(* IEC 61131-3 sources: Temperature-Cabinet-Control-Automation/codesys modbus proof of concept and test logs/src/POUs, 2 files *)

(* ---- PLC_PRG.st ---- *)
(*
    PROGRAM:  PLC_PRG
    Project:  Temperature Cabinet Setpoint Control from CODESYS HMI
    Author:   OJ (Omkar Joshi) - Oliver Mechatronics
    Language: IEC 61131-3 Structured Text (CODESYS 3.5, WebVisu)

    Cyclic entry point (MainTask). Instantiates the supervisory setpoint
    controller. Because FB_CabinetSetpointControl reads/writes GVL_Modbus
    and GVL_HMI directly in its body (see that FB's header note), this
    program only needs to pass through the operator-facing parameters
    and the safety interlock input.

    Matches the Project Development Package spec (Details A) and the
    build guide already in codesys modbus com port investigation and troubleshooting log/README.md.

    TODO (flagged in the Project Development Package, not yet resolved):
    xOverTempDI below is wired to GVL_Modbus.xModbusError as a
    placeholder. REPLACE with the real mapped EL1409 digital-input
    channel (spare over-temperature lamp contact) in the EtherCAT I/O
    mapping before relying on this interlock.
*)
PROGRAM PLC_PRG
VAR
    fbSetpoint : FB_CabinetSetpointControl;
END_VAR

(* ---- Drive the supervisory setpoint controller ---- *)
fbSetpoint(
    rRequestedSetpoint := GVL_HMI.rReqSetpoint,
    xSetCommand        := GVL_HMI.xSetBtn,
    xReset             := GVL_HMI.xResetBtn,
    xOverTempDI        := GVL_Modbus.xModbusError,  (* REPLACE with mapped EL1409 DI channel *)
    rMinSetpoint       := -40.0,
    rMaxSetpoint       := 200.0
);

(* ---- Consume dialog button one-shots ---- *)
GVL_HMI.xSetBtn   := FALSE;
GVL_HMI.xResetBtn := FALSE;

(* ---- PLC_PRG_TCP.st ---- *)
PROGRAM PLC_PRG
(* ======================================================================
   Retargeted for TCP register sources (Python gateway via Modbus TCP)
   ======================================================================
   Serial device abandoned. All reads/writes now come via the TCP slave
   device on the Modbus TCP master branch of the device tree.

   Proven register map (TCP holding registers, x10 integers):
     reg2 = chamber temperature (read-only, cyclic)
     reg3 = confirmed setpoint read-back (read-only, cyclic)
     reg4 = status/fault code (read-only, cyclic)
     reg0 = requested setpoint (write, cyclic or rising)
     reg1 = apply trigger (write, rising edge)

   I/O Mapping binds these to GVL_Modbus:
     reg2 -> wInput1Value (temperature)
     reg3 -> wSetpoint1Read (confirmed SP)
     reg4 -> wStatus (fault code: 0=OK, 2=WRITE_FAILED, 3=NOT_ACCEPTED, 4=RANGE, 5=COMMS)
     reg0 -> wSetpoint1Write (requested SP, x10)
     reg1 -> xWriteTrigger (apply pulse, BOOL as WORD 0/1)

   The state machine logic is unchanged from the serial version. Only the
   data sources changed: TCP channels instead of serial channels.
   ====================================================================== *)

VAR
    rChamberTemp        : REAL;
    rReqSetpoint        : REAL := 26.5;           (* set in watch window or WebVisu *)
    rConfirmedSetpoint  : REAL;

    rMinSetpoint        : REAL := -40.0;
    rMaxSetpoint        : REAL := 200.0;

    eSetpointState      : E_SetpointState := E_SetpointState.IDLE;
    eFaultCode          : E_FaultCode := E_FaultCode.NO_FAULT;

    xStartWrite         : BOOL := FALSE;          (* rising-edge trigger for manual test *)
    xPrevStartWrite     : BOOL := FALSE;
    xWriteTriggered     : BOOL := FALSE;

    dwWriteTimeout      : DWORD := 0;
    (* Must exceed the WORST-CASE confirm chain, not the typical one:
         gateway poll period            1.0 s   (POLL_PERIOD)
       + gateway RTU confirm read-back  0.5 s   (READ_TIMEOUT)
       + CODESYS cyclic read of reg3    2.0 s   (channel 3 trigger interval)
       = 3.5 s worst case, against a 3.0 s timeout -> spurious NOT_ACCEPTED on
       a write the F4S had actually taken. Raised to 10 s so only a genuine
       failure trips it; the gateway's own status codes (2/3/5) still fault
       fast, so a real rejection is never delayed by this headroom. *)
    dwMaxTimeout        : DWORD := 1000;          (* ~10s at 10ms MainTask *)

    dtNow               : DT;                      (* current local time for schedule *)
    uliHighRes          : ULINT;                   (* high-resolution time, raw ms since epoch, UTC *)
END_VAR

(* --- STEP 0: Cabinet on/off - EL2869 CH15/CH16 -> Omron CPM1A digital inputs ---
   AS-BUILT 6 Aug 2026 (README §19), supersedes the §17 F4-DI ramp gate for on/off.
   CH15 -> wire 102 -> Omron 0CH.00 (start input to the Omron's own start-stop-hold
   ladder logic). CH16 -> wire 103 -> Omron 0CH.01 (stop input). EL2869 DO GND is
   bonded to Omron COM0.

   xStartPulse and xStopPermit are plain, independently-commanded levels -- no
   timer, no derived pulse, no anti-short-cycle lockout. Set them from the watch
   window (or, later, WebVisu) and they hold until changed. The Omron's own
   program does the actual start-stop-hold latching, so CODESYS only needs to
   present a level on each input; it does not need to shape a pulse width the way
   the earlier (§15 Option C-era) design did.

   That earlier design drove xStartPulse off a TP one-shot fired on the rising
   edge of xStopPermit, modelling CH16 as a continuous 24 V supply that CH15
   briefly "pressed" through (the button-station supply-lift model). That model
   does not apply to the Omron's digital inputs and is what produced the reported
   "stop permit true, then false, then start pulse fires" sequence -- an artifact
   of the old coupling, not the Omron's behaviour. Removed here.

   The only guard kept in is stop-priority mutual exclusion: if both are ever
   commanded TRUE together, stop wins. This costs one line and there is no
   scenario where firing both at once is the intended action -- flag it for
   removal if that turns out to be unwanted.

   xCabinetOnCmd (scheduler-derived, below) is NOT wired into xStartPulse/
   xStopPermit yet -- open question, README §19, on whether the schedule should
   auto-drive start/stop or these should stay purely operator/CODESYS-commanded. *)
SysTimeRtcHighResGet(uliHighRes);
dtNow := ULINT_TO_DT(uliHighRes / 1000 + DINT_TO_ULINT(GVL_HMI.diUtcOffsetSec));  (* ms -> s, then UTC -> local *)

GVL_HMI.xCabinetOnCmd := NOT (GVL_HMI.xSchedEnable AND (dtNow < GVL_HMI.dtSchedStart));

IF GVL_HMI.xStopPermit THEN
    GVL_HMI.xStartPulse := FALSE;
END_IF

GVL_HMI.xCabinetRunning := GVL_HMI.xStartPulse AND NOT GVL_HMI.xStopPermit;  (* commanded-state
    proxy for WebVisu -- no independent run feedback wired back from the Omron yet, README §19.6 *)

(* --- STEP 0b: Front-panel keypad lock (§17/§18 F4 digital input design) ---
   NOT CURRENTLY WIRED. CH16 is now committed to the Omron stop input above, so
   xPanelLock has no live output channel until §18's D/I 2 is reallocated to a
   spare EL2869 channel (README §19.5). Left commented out rather than deleted so
   the logic is ready to reconnect once that channel is chosen and mapped:

   GVL_HMI.xPanelLock := GVL_HMI.xPanelLockCmd;
*)

(* --- STEP 1: Scale raw TCP values -> engineering units ---
   TCP registers carry x10 integers; we work in real degrees.
   All three reads come from the TCP channels (wInput1Value, wSetpoint1Read, wStatus).

   The registers carry SIGNED x10 integers in two's complement. WORD is an
   UNSIGNED type in IEC 61131-3, so dividing it directly turns -1.0 degC
   (raw 16#FFF6) into 6552.6 instead of -1.0. Every sub-zero temperature and
   every negative setpoint read-back was wrong, and the CONFIRM comparison
   below could never match one. WORD_TO_INT reinterprets the bit pattern as
   the signed value the F4S actually sent.
*)
rChamberTemp       := WORD_TO_INT(GVL_Modbus.wInput1Value)  / 10.0;
rConfirmedSetpoint := WORD_TO_INT(GVL_Modbus.wSetpoint1Read) / 10.0;

(* --- STEP 2: Detect rising edge on the manual test trigger ---
   When testing from watch window, toggle xStartWrite from FALSE to TRUE.
   In production (WebVisu or SCADA), the operator triggers via a button that
   sets a HMI variable, but the edge logic is the same.
*)
xWriteTriggered := (xStartWrite AND NOT xPrevStartWrite);
xPrevStartWrite := xStartWrite;

(* --- STEP 3: State machine (unchanged logic, TCP-based register sources) --- *)

CASE eSetpointState OF

    E_SetpointState.IDLE:
        (* Waiting for a write request. Hold the apply trigger low. *)
        GVL_Modbus.xWriteTrigger := FALSE;
        dwWriteTimeout := 0;

        IF xWriteTriggered THEN
            eSetpointState := E_SetpointState.READY;
        END_IF

    E_SetpointState.READY:
        (* Validate the requested setpoint against limits. *)
        IF rReqSetpoint < rMinSetpoint THEN
            eFaultCode := E_FaultCode.RANGE_LOW;
            eSetpointState := E_SetpointState.FAULTED;

        ELSIF rReqSetpoint > rMaxSetpoint THEN
            eFaultCode := E_FaultCode.RANGE_HIGH;
            eSetpointState := E_SetpointState.FAULTED;

        ELSE
            (* Valid range. Stage the request (x10 int) into the TCP write register.

               REAL_TO_DWORD is UNDEFINED for negative operands in IEC 61131-3
               -- it happened to produce the right bit pattern on this runtime,
               but that is luck, not contract, and it truncates instead of
               rounding (26.45 -> 264, not 265). REAL_TO_INT rounds and is
               defined across the whole -40..200 range; INT_TO_WORD then
               reinterprets the signed value as the two's-complement WORD the
               gateway expects on the wire. *)
            GVL_Modbus.wSetpoint1Write := INT_TO_WORD(REAL_TO_INT(rReqSetpoint * 10.0));
            eSetpointState := E_SetpointState.WRITING;
        END_IF

    E_SetpointState.WRITING:
        (* Pulse the apply trigger (one scan). The Python gateway services this
           by writing reg1=1 over RTU and then clearing it to 0 when done. *)
        GVL_Modbus.xWriteTrigger := TRUE;
        dwWriteTimeout := 0;
        eSetpointState := E_SetpointState.CONFIRM;

    E_SetpointState.CONFIRM:
        (* Drop the trigger immediately to re-arm the edge for the next request. *)
        GVL_Modbus.xWriteTrigger := FALSE;
        dwWriteTimeout := dwWriteTimeout + 1;

        (* Check for immediate comms failure (Python gateway lost). *)
        IF GVL_Modbus.wStatus = 5 THEN                  (* COMMS fault from gateway *)
            eFaultCode := E_FaultCode.COMMS_TIMEOUT;
            eSetpointState := E_SetpointState.FAULTED;

        (* Check for write-accepted confirmation: read-back matches request. *)
        ELSIF ABS(rConfirmedSetpoint - rReqSetpoint) < 0.1 THEN
            eFaultCode := E_FaultCode.NO_FAULT;
            eSetpointState := E_SetpointState.IDLE;

        (* Check for write-failed fault (Python couldn't write to F4S). *)
        ELSIF GVL_Modbus.wStatus = 2 THEN                (* WRITE_FAILED *)
            eFaultCode := E_FaultCode.WRITE_FAILED;
            eSetpointState := E_SetpointState.FAULTED;

        (* Check for not-accepted fault (F4S silent-rejected, e.g., menu mode). *)
        ELSIF GVL_Modbus.wStatus = 3 THEN                (* NOT_ACCEPTED *)
            eFaultCode := E_FaultCode.NOT_ACCEPTED;
            eSetpointState := E_SetpointState.FAULTED;

        (* Check for range/fault from Python side.
           The gateway reports a single RANGE code (4) without a direction, so
           resolve LOW vs HIGH from the request we actually sent. Reporting
           every gateway range reject as RANGE_HIGH sent the operator hunting
           for a ceiling problem when a -1.0 degC request had tripped the
           gateway's old unsigned 0..2000 check at the FLOOR. *)
        ELSIF GVL_Modbus.wStatus = 4 THEN                (* RANGE *)
            IF rReqSetpoint < rMinSetpoint THEN
                eFaultCode := E_FaultCode.RANGE_LOW;
            ELSE
                eFaultCode := E_FaultCode.RANGE_HIGH;
            END_IF
            eSetpointState := E_SetpointState.FAULTED;

        (* Timeout: Python didn't respond in time. *)
        ELSIF dwWriteTimeout > dwMaxTimeout THEN
            eFaultCode := E_FaultCode.NOT_ACCEPTED;      (* treated as F4S rejection *)
            eSetpointState := E_SetpointState.FAULTED;
        END_IF

    E_SetpointState.FAULTED:
        (* Latched fault state. User must acknowledge by re-triggering (watch window or HMI). *)
        GVL_Modbus.xWriteTrigger := FALSE;

        IF xWriteTriggered THEN
            eFaultCode := E_FaultCode.NO_FAULT;
            eSetpointState := E_SetpointState.READY;
        END_IF

END_CASE

(* --- STEP 4: Consume the manual test trigger (so it doesn't re-fire) ---
   In production, replace xStartWrite with the HMI/WebVisu button signal.
   The gateway's apply trigger (reg1) is cleared by the Python side after processing.
*)
xStartWrite := FALSE;
